TYPE TestCaseHandle_t : POINTER TO FB_UnitTestBase; END_TYPE

(* stored: Version 1.1.0.1, ProductVersion 3.1.4022.9
   DUT TestCaseHandle_t: Id {ddf66e01-3edf-4aca-b370-8d31156ec1d8} *)
